FUNCTION F_AnalogScale : INT
VAR_INPUT
	AnalogInputRawValue	: DINT;
	MaxAnalogValue		: INT;
END_VAR
VAR
	MaxInput			: INT;
	ScaledValue: INT;
END_VAR
VAR_OUTPUT
END_VAR

// 4-20 mA: 0-32767
MaxInput := 32767;
F_AnalogScale := REAL_TO_INT(AnalogInputRawValue / (MaxInput / MaxAnalogValue));

END_FUNCTION

(* stored: Version 1.1.0.1, ProductVersion 3.1.4024.9
   POU F_AnalogScale: Id {ede14f80-1557-42a5-a2f9-8ca8f4e9e338}, SpecialFunc None *)
